{attribute addProperty BoxType "KL1002"}
{attribute addProperty Id "InputAT %I*BOOL000"}
{attribute addProperty CRC "1890977489"}
{attribute addProperty SizeInBites "0"}
{attribute addProperty SizeInBytes "0"}
TYPE Channel_70B606D1 :
STRUCT
	{attribute addProperty Name "Input"}
	Input AT %I* : BOOL;
END_STRUCT
END_TYPE

(* stored: Version 1.2.0.0, ProductVersion 3.1.4024.9
   DUT Channel_70B606D1: Id {00dd0e73-e40e-4e2a-941d-a70e734d72bf} *)
